{attribute addProperty BoxType "EL6001-0000-0020"}
{attribute addProperty Id "StatusAT %I*Status_A3013EBE8Data_InAT %I*ARRAY[0..21] OF USINT22"}
{attribute addProperty CRC "3350509587"}
{attribute addProperty SizeInBites "240"}
{attribute addProperty SizeInBytes "30"}
TYPE COM_Inputs_F2FBC98A :
STRUCT
	{attribute addProperty Name "Status"}
	Status AT %I* : Status_A3013EBE;
	{attribute addProperty Name "Data_In"}
	Data_In AT %I* : ARRAY[0..21] OF USINT;
END_STRUCT
END_TYPE

(* stored: Version 1.2.0.0, ProductVersion 3.1.4024.9
   DUT COM_Inputs_F2FBC98A: Id {61bdc687-eeb1-4e4e-91b2-cb8ee86f7c53} *)
